FUNCTION F_LRealToString : STRING(255)
VAR_INPUT
	fValue: LREAL;
END_VAR

F_LRealToString := F_LRealToStringEx(fValue, 3);

END_FUNCTION

(* stored: Version 1.1.0.1, ProductVersion 3.1.4022.9
   POU F_LRealToString: Id {893b7018-a3d0-49a4-a7c2-880be2b53ec0}, SpecialFunc None *)
